// TIA Portal V18 export
FUNCTION_BLOCK "TD_Motor_Start_CAT"   // FB14, LAD
{ S7_Optimized_Access := 'TRUE' }
// Written BY Kristopher Gimenez January 25,2023
// This block is used to control the Aux, and Cooler fan motors.
// stored: AutoNumber false, MemoryReserve 100, SetENOAutomatically false
   VAR
      EngineFault_TON { S7_SetPoint := 'True'} : TON_TIME;
   END_VAR
   VAR_TEMP
      tempReal : Real;
   END_VAR
BEGIN

REGION Network 1: Engine Speed
   // Pulse Per Second X 60sc/m /PPR
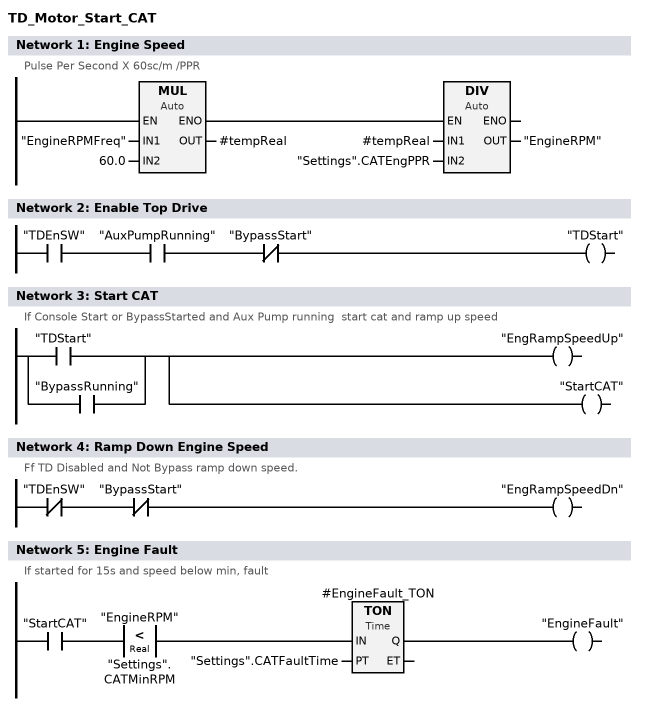
   RUNG wire#powerrail
      Mul(in1 := "EngineRPMFreq", in2 := 60.0, out => #tempReal)
      Div(in1 := #tempReal, in2 := "Settings".CATEngPPR, out => "EngineRPM")
   END_RUNG
   // the same network as SCL:
   #tempReal := "EngineRPMFreq" * 60.0;
   "EngineRPM" := #tempReal / "Settings".CATEngPPR;
END_REGION

REGION Network 2: Enable Top Drive
   RUNG wire#powerrail
      Contact( "TDEnSW" )
      Contact( "AuxPumpRunning" )
      I_Contact( "BypassStart" )
      Coil( "TDStart" )
   END_RUNG
   // the same network as SCL:
   "TDStart" := "TDEnSW" AND "AuxPumpRunning" AND NOT "BypassStart";
END_REGION

REGION Network 3: Start CAT
   // If Console Start or BypassStarted and Aux Pump running  start cat and ramp up speed
   RUNG wire#powerrail
      Contact( "TDStart" )
      wire#w1
      Coil( "EngRampSpeedUp" )
   END_RUNG
   RUNG wire#powerrail
      Contact( "BypassRunning" )
   END_RUNG wire#w1
   RUNG wire#w1
      Coil( "StartCAT" )
   END_RUNG
   // the same network as SCL:
   "EngRampSpeedUp" := "TDStart" OR "BypassRunning";
   "StartCAT" := "EngRampSpeedUp";
END_REGION

REGION Network 4: Ramp Down Engine Speed
   // Ff TD Disabled and Not Bypass ramp down speed.
   RUNG wire#powerrail
      I_Contact( "TDEnSW" )
      I_Contact( "BypassStart" )
      Coil( "EngRampSpeedDn" )
   END_RUNG
   // the same network as SCL:
   "EngRampSpeedDn" := NOT "TDEnSW" AND NOT "BypassStart";
END_REGION

REGION Network 5: Engine Fault
   // If started for 15s and speed below min, fault
   RUNG wire#powerrail
      Contact( "StartCAT" )
      { S7_Templates := "SrcType := Real" } LT_Contact(in1 := "EngineRPM", in2 := "Settings".CATMinRPM)
      { S7_Templates := "time_type := Time" } #EngineFault_TON.TON(pt := "Settings".CATFaultTime, et =>)
      Coil( "EngineFault" )
   END_RUNG
   // the same network as SCL:
   #EngineFault_TON(IN := "StartCAT" AND ("EngineRPM" < "Settings".CATMinRPM), PT := "Settings".CATFaultTime);   // TON
   "EngineFault" := #EngineFault_TON.Q;
END_REGION
END_FUNCTION_BLOCK
